TYPE ESR_DATA :
STRUCT
	TYP : BYTE;
	ADRESS : STRING(10);
	DS : DT;
	TS : TIME;
	DATA : ARRAY[0..7] OF BYTE;
END_STRUCT
END_TYPE

(* stored: Version 1.1.0.1
   DUT ESR_DATA: Id {d8e1cda0-c8b4-42cc-a322-b2403c1fa8c8} *)
